(* PLC project beckhoff_vision, Institute of Astronomy Onto 0.0.1 *)
(* stored: creationDateTime 2025-01-01T00:00:00.0, modificationDateTime 2025-01-01T00:00:00.0 *)

TYPE ETcVnCameraState : (TCVN_CS_ERROR := 0, TCVN_CS_INITIAL := 1, TCVN_CS_INITIALIZING := 2, TCVN_CS_INITIALIZED := 3, TCVN_CS_OPENING := 4, TCVN_CS_OPENED := 5, TCVN_CS_STARTACQUISITION := 6, TCVN_CS_ACQUIRING := 7, TCVN_CS_STOPACQUISITION := 8, TCVN_CS_RESETTINGFEATURES := 9, TCVN_CS_TRIGGERING := 10, TCVN_CS_CLOSING := 11);
END_TYPE
